# B&R Automation Studio project mappCfg
Automation Studio 4.9.3.144 SP; technology packages: mapp 5.15.0

## Configuration Config1

CPU X20CP3585, AutomationRuntime D4.90, Build 4.1.2, Safety 0.0, Vc V4.72.6

### Task classes (Cpu.sw)
```
Cyclic#4:
  MpLinkTest <- (binary)
Cyclic#8:
  MpCfgTest <- MpCfgTest.prg
Binaries: FWRules, udbdef, arsvcreg, TCData, User, arconfig, Role, Config, iomap, asfw, ashwac, ashwd, sysconf
Libraries: MpCom, MpBase, MpCfg, FileIO, runtime, astime, asieccon, AsBrStr, IecCheck, sys_lib, MpUserX
```

### Hardware
```
X20CP3585 : X20CP3585 v1.10.0.0
  Connector IF2:
    ActivateDevice = 1
  ConfigurationID = mappLink_Config1
  FtpUser1
  FtpUsername1 = bur
  FtpUserPassword1 = 9h9s1YQ4rmHMniR3mwrIYznV2yRb7wj1AtHiJ/RHOmI=  // bur
  FtpUserSalt1 = llDQoh2a
  FTPAccessRight1 = 0
  FTPMSPartition1 = SYSTEM
```

### Config.mpdatabasecore - X20CP3585/mappServices/Config.mpdatabasecore
```
Element gDatabaseCore (Type=mpdatabasecore)
  mapp.Database.Core:
    Name = brdatabase
    UserName = br
    Password = bandr
    IPAddress  // IPv4 address of the database script
    PortNumber = 85  // SQL port number of the database script
    DBQueries:
      [0]:
        Name = RecipeLoad
        Type:
          Select:
            Columns:
              PV = ::Recipe.DATA
          From = dbo.brtable
          Where:
            [0]:
              Column = product_name
              Operator = eq
              CompareTo:
                Value = {&pv[Recipe.PAR.RecipeName]}
      [1]:
        Name = RecipeSave
        Type:
          1TypeName = UPDATE
          Where:
            [0]:
              Column = product_name
              Operator = eq
              CompareTo:
                Value = {&pv[Recipe.PAR.RecipeName]}
      [2]:
        Name = RecipeDelete
        Type:
          1TypeName = DELETE
          Where:
            [0]:
              Column = product_name
              Operator = eq
              CompareTo:
                Value = {&pv[Recipe.PAR.RecipeName]}
      [3]:
        Name = RecipeNew
        Type:
          1TypeName = INSERT
      [4]:
        Name = RecipeList
        Type:
          1TypeName = Custom
```

### Config_1.mpuserx - X20CP3585/mappServices/Config_1.mpuserx
```
Element UserMgmtX (Type=mpuserx)
  ServerSettings:
    Server:
      AdditionalUserData:
        [0] = mail
        [1] = telephoneNumber
  Users:
    DefUser#1:
      id = Anonymous
      name = Nobody
    DefUser#2:
      id = John
      name = John Doe
    DefUser#3:
      id = Jane
      name = Jane Doe
```

## Logical view

Binary libraries used (declarations not repeated): operator, runtime, astime, AsIecCon, FileIO, AsBrStr, IecCheck, sys_lib, MpCom, MpBase, MpUserX 5.15.0

### Package Logical/Libraries - Global libraries

### Library Logical/Libraries/MpCfg (IEC)

#### Types.typ - Exported data types
```iecst
TYPE
	MpCfgInfoType : 	STRUCT
		state : MpCfgStateType;
		DevLink_1 : DevLink;
		FileOpen_1 : FileOpen;
		FileRead_1 : FileRead;
		FileWrite_1 : FileWrite;
		FileClose_1 : FileClose;
		MpComConfigManager_1 : MpComConfigManager;
		Buffer : ARRAY[0..MpCfgMaxBufferSize]OF USINT;
		NodeName : STRING[MpCfgMaxNameSize];
		NodeValue : STRING[MpCfgMaxValueSize];
		offset1 : DINT;
		offset2 : DINT;
		len : DINT;
		tmpStr1 : STRING[MpCfgMaxNameSize];
		tmpStr2 : STRING[MpCfgMaxNameSize];
	END_STRUCT;
	MpCfgStateType :
		(
		stateWait,
		stateDevLink,
		stateExport,
		stateOpen,
		stateRead,
		stateWrite,
		stateClose,
		stateFindData,
		stateInsertData,
		stateError
		);
END_TYPE
```

#### Constants.var - Exported constants
```iecst
(*Buffer and variable sizes*)
VAR CONSTANT
	MpCfgMaxBufferSize : UINT := 10000;
	MpCfgMaxNameSize : UINT := 200;
	MpCfgMaxValueSize : UINT := 200;
END_VAR
(*Error numbers*)
VAR CONSTANT
	MpCfgBufferSizeExceeded : DINT := 10001;
	MpCfgDataTypeSizeExceeded : DINT := 10002;
	MpCfgValueSizeExceeded : DINT := 10003;
	MpCfgGroupNotFound0 : DINT := 10010;
	MpCfgGroupNotFound1 : DINT := 10011;
	MpCfgGroupNotFound2 : DINT := 10012;
	MpCfgGroupNotFound3 : DINT := 10013;
	MpCfgGroupNotFound4 : DINT := 10014;
	MpCfgGroupNotFound5 : DINT := 10015;
	MpCfgGroupNotFound6 : DINT := 10016;
	MpCfgGroupNotFound7 : DINT := 10017;
	MpCfgGroupNotFound8 : DINT := 10018;
	MpCfgGroupNotFound9 : DINT := 10019;
	MpCfgParaNotFound : DINT := 10020;
	MpCfgTypeNotFound : DINT := 10021;
	MpCfgValueNotFound : DINT := 10022;
	MpCfgParaNameEmpty : DINT := 10030;
	MpCfgMpLinkEmpty : DINT := 10031;
END_VAR
(*Read/Write constants*)
VAR CONSTANT
	MpCfgRead : BOOL := FALSE;
	MpCfgWrite : BOOL := TRUE;
END_VAR
```

#### MpCfg.fun - Exported functions and function blocks
```iecst
FUNCTION_BLOCK MpCfgRW
	VAR_INPUT
		MpLink : {REDUND_UNREPLICABLE} MpComIdentType;
		Enable : BOOL;
		ReadWrite : BOOL;
		ErrorReset : BOOL;
		ParaName : STRING[MpCfgMaxNameSize];
		ParaValue : STRING[MpCfgMaxValueSize];
	END_VAR
	VAR_OUTPUT
		Active : BOOL;
		Error : BOOL;
		StatusID : DINT;
		CommandDone : BOOL;
		DataType : STRING[50];
		Value : STRING[MpCfgMaxValueSize];
	END_VAR
	VAR
		Info : MpCfgInfoType;
	END_VAR
END_FUNCTION_BLOCK

FUNCTION FindInMem : DINT
	VAR_INPUT
		data1 : UDINT;
		len1 : UDINT;
		data2 : UDINT;
		len2 : UDINT;
		direction : BOOL;
	END_VAR
	VAR
		idx : UDINT;
	END_VAR
END_FUNCTION

FUNCTION ReplaceString : BOOL
	VAR_INPUT
		dataSTR : UDINT;
		searchSTR : UDINT;
		replaceSTR : UDINT;
		first : BOOL;
	END_VAR
	VAR
		idx : UDINT;
	END_VAR
END_FUNCTION
```

#### MpCfg.st
```iecst
// -------------------------------------------------------------------------
// Read mapp configuration parameter
// -------------------------------------------------------------------------
FUNCTION_BLOCK MpCfgRW
	// Abort command
	IF EDGENEG(Enable) THEN
		// Close file if it was already opened
		IF Info.state >= stateOpen AND Info.state <> stateError THEN
			Info.state := stateClose;
		END_IF
	END_IF

	// -------------------------------------------------------------------------
	// MpLink state machine
	CASE Info.state OF
		// -------------------------------------------------------------------------
		// Wait for new command
		stateWait:
			// Reset all funtion blocks
			Info.DevLink_1.enable 				:= FALSE;
			Info.DevLink_1();
			Info.MpComConfigManager_1.Enable 	:= FALSE;
			Info.MpComConfigManager_1();
			Info.FileOpen_1.enable				:= FALSE;
			Info.FileOpen_1();
			Info.FileRead_1.enable				:= FALSE;
			Info.FileRead_1();
			Info.FileClose_1.enable				:= FALSE;
			Info.FileClose_1();

			// New command
			IF EDGEPOS(Enable) THEN
				// Make sure MpLink is not empty
				IF MpLink.Internal[0] = 0 THEN
					StatusID := MpCfgMpLinkEmpty;
					Info.state := stateError;
				ELSE
					// Make sure parameter is not empty
					IF ParaName = '' THEN
						StatusID := MpCfgParaNameEmpty;
						Info.state := stateError;
					ELSE
						// Set start values
						Active := TRUE;
						DataType := '';
						Value := '';
						brsmemset(ADR(Info.Buffer), 0, SIZEOF(Info.Buffer));
						Info.state := stateDevLink;
					END_IF
				END_IF
			ELSE
				IF NOT Enable THEN
					CommandDone := FALSE;
				END_IF
				Active := FALSE;
			END_IF
			// -------------------------------------------------------------------------
		// Link file device used for exporting data
		stateDevLink:
			Info.DevLink_1.enable 	:= TRUE;
			Info.DevLink_1.pDevice	:= ADR('MpCfgDev');
			Info.DevLink_1.pParam	:= ADR('/DEVICE=C:/');
			Info.DevLink_1();

			// Success
			IF Info.DevLink_1.status = ERR_OK OR Info.DevLink_1.status = fiERR_DEVICE_ALREADY_EXIST THEN
				Info.state := stateExport;
			// Errror
			ELSIF Info.DevLink_1.status <> ERR_FUB_BUSY THEN
				StatusID := Info.DevLink_1.status;
				Info.state := stateError;
			END_IF
		// -------------------------------------------------------------------------
		// Export mapp data
		stateExport:
			Info.MpComConfigManager_1.Enable 		:= TRUE;
			Info.MpComConfigManager_1.MpLink		:= ADR(MpLink);
			Info.MpComConfigManager_1.DeviceName 	:= ADR('MpCfgDev');
			Info.MpComConfigManager_1.FileName 		:= ADR('MpCfg.xml');
			Info.MpComConfigManager_1.Scope			:= mpCOM_CONFIG_SCOPE_COMPONENT;
			Info.MpComConfigManager_1.Export		:= TRUE;
			Info.MpComConfigManager_1.Import		:= FALSE;
			Info.MpComConfigManager_1();

			// Success
			IF Info.MpComConfigManager_1.CommandDone AND NOT Info.MpComConfigManager_1.Error THEN
				Info.state := stateOpen;
			// Errror
			ELSIF Info.MpComConfigManager_1.Error THEN
				StatusID := Info.MpComConfigManager_1.StatusID;
				Info.state := stateError;
			END_IF
		// -------------------------------------------------------------------------
		// Open mapp data
		stateOpen:
			Info.FileOpen_1.enable		:= TRUE;
			Info.FileOpen_1.pDevice 	:= ADR('MpCfgDev');
			Info.FileOpen_1.pFile		:= ADR('MpCfg.xml');
			Info.FileOpen_1.mode 		:= fiREAD_WRITE;
			Info.FileOpen_1();

			// Success
			IF Info.FileOpen_1.status = ERR_OK THEN
				IF Info.FileOpen_1.filelen > SIZEOF(Info.Buffer) THEN
					StatusID := MpCfgBufferSizeExceeded;
					Info.state := stateError;
				ELSE
					Info.state := stateRead;
				END_IF
			// Errror
			ELSIF Info.FileOpen_1.status <> ERR_FUB_BUSY THEN
				StatusID := Info.FileOpen_1.status;
				Info.state := stateError;
			END_IF

		// -------------------------------------------------------------------------
		// Read mapp data file
		stateRead:
			Info.FileRead_1.enable		:= TRUE;
			Info.FileRead_1.ident		:= Info.FileOpen_1.ident;
			Info.FileRead_1.len			:= Info.FileOpen_1.filelen;
			Info.FileRead_1.pDest		:= ADR(Info.Buffer);
			Info.FileRead_1();

			// Success
			IF Info.FileRead_1.status = ERR_OK THEN
				// Find group id first
				IF ADR(GroupArray) <> 0 THEN
					// Make sure array has at least one entry
					IF GroupArray.Item[0] <> '' THEN
						Info.idx := 0;
						Info.DataOffset1 := 0;
						Info.state := stateFindGroup;
					// Find unique parameter
					ELSE
						Info.state := stateFindData;
					END_IF
				// Find unique parameter
				ELSE
					Info.state := stateFindData;
				END_IF
			// Errror
			ELSIF Info.FileRead_1.status <> ERR_FUB_BUSY THEN
				StatusID := Info.FileRead_1.status;
				Info.state := stateError;
			END_IF

		// -------------------------------------------------------------------------
		// Write mapp data file
		stateWrite:
			Info.FileWrite_1.enable		:= TRUE;
			Info.FileWrite_1.ident		:= Info.FileOpen_1.ident;
			Info.FileWrite_1.len		:= Info.FileLen;
			Info.FileWrite_1.pSrc		:= ADR(Info.Buffer);
			Info.FileWrite_1();

			// Success
			IF Info.FileWrite_1.status = ERR_OK THEN
				Info.state := stateClose;
			// Errror
			ELSIF Info.FileWrite_1.status <> ERR_FUB_BUSY THEN
				StatusID := Info.FileWrite_1.status;
				Info.state := stateError;
			END_IF

		// -------------------------------------------------------------------------
		// Find group data
		stateFindGroup:
			// Prepare group string
			Info.tmpStr1 := '<Group ID="';
			brsstrcat(ADR(Info.tmpStr1), ADR(GroupArray.Item[Info.idx]));
			brsstrcat(ADR(Info.tmpStr1), ADR('"'));
			// Find property string
			Info.DataOffset1 := Info.DataOffset1+FindInMem(ADR(Info.Buffer)+Info.DataOffset1, Info.FileOpen_1.filelen, ADR(Info.tmpStr1), brsstrlen(ADR(Info.tmpStr1)), FALSE);

			// Found group string
			IF Info.DataOffset1 > -1 THEN
				// Find next group name
				IF Info.idx < SIZEOF(GroupArray)/SIZEOF(GroupArray.Item[0]) THEN
					Info.idx := Info.idx + 1;
					IF GroupArray.Item[Info.idx] = '' THEN
						Info.state := stateFindData;
					END_IF
				// Group was not found
				ELSE
					StatusID := MpCfgGroupNotFound0+Info.idx;
					Info.state := stateError;
				END_IF
			// Group was not found
			ELSE
				StatusID := MpCfgGroupNotFound0+Info.idx;
				Info.state := stateError;
			END_IF
		// -------------------------------------------------------------------------
		// Find data
		stateFindData:
			// Prepare property string
			Info.tmpStr1 := '<Property ID="';
			brsstrcat(ADR(Info.tmpStr1), ADR(ParaName));
			brsstrcat(ADR(Info.tmpStr1), ADR('"'));
			// Find property string
			Info.DataOffset1 := Info.DataOffset1+FindInMem(ADR(Info.Buffer)+Info.DataOffset1, Info.FileOpen_1.filelen, ADR(Info.tmpStr1), brsstrlen(ADR(Info.tmpStr1)), FALSE);

			// Found parameter string
			IF Info.DataOffset1 > -1 THEN
				// Prepare data type start string
				Info.tmpStr1 := 'DataType="';
				// Find data type string start
				Info.DataOffset2 := brsstrlen(ADR(Info.tmpStr1))+FindInMem(ADR(Info.Buffer)+Info.DataOffset1, Info.FileOpen_1.filelen, ADR(Info.tmpStr1), brsstrlen(ADR(Info.tmpStr1)), FALSE);

				// Found data type start
				IF Info.DataOffset2 > -1 THEN
					// Prepare data type end string
					Info.tmpStr1 := '"';
					// Find data type string
					Info.DataLen := FindInMem(ADR(Info.Buffer)+Info.DataOffset1+Info.DataOffset2, Info.FileOpen_1.filelen, ADR(Info.tmpStr1), brsstrlen(ADR(Info.tmpStr1)), FALSE);

					// Found data type end, copy data to output
					IF Info.DataLen > -1 THEN
						brsmemset(ADR(DataType), 0, SIZEOF(DataType));
						brsmemcpy(ADR(DataType), ADR(Info.Buffer)+Info.DataOffset1+Info.DataOffset2, Info.DataLen);

						// Prepare value start string
						Info.tmpStr1 := 'Value="';
						// Find data type string start
						Info.DataOffset2 := brsstrlen(ADR(Info.tmpStr1))+FindInMem(ADR(Info.Buffer)+Info.DataOffset1, Info.FileOpen_1.filelen, ADR(Info.tmpStr1), brsstrlen(ADR(Info.tmpStr1)), FALSE);

						// Found value start
						IF Info.DataOffset2 > -1 THEN
							// Prepare value end string
							Info.tmpStr1 := '"';
							// Find value end string
							Info.DataLen := FindInMem(ADR(Info.Buffer)+Info.DataOffset1+Info.DataOffset2, Info.FileOpen_1.filelen, ADR(Info.tmpStr1), brsstrlen(ADR(Info.tmpStr1)), FALSE);

							// Found value end, copy data to output
							IF Info.DataLen > -1 THEN
								brsmemset(ADR(Value), 0, SIZEOF(Value));
								brsmemcpy(ADR(Value), ADR(Info.Buffer)+Info.DataOffset1+Info.DataOffset2, Info.DataLen);

								// Finish when command is reading
								IF ReadWrite = MpCfgRead THEN
									Info.state := stateClose;
								// Insert new data in next step
								ELSE
									Info.state := stateInsertData;
								END_IF
							// Value end was not found
							ELSE
								StatusID := MpCfgValueNotFound;
								Info.state := stateError;
							END_IF
						// Value start was not found
						ELSE
							StatusID := MpCfgValueNotFound;
							Info.state := stateError;
						END_IF
					// Data type end was not found
					ELSE
						StatusID := MpCfgTypeNotFound;
						Info.state := stateError;
					END_IF
				// Data type end was not found
				ELSE
					StatusID := MpCfgTypeNotFound;
					Info.state := stateError;
				END_IF
			// Parameter name was not found
			ELSE
				StatusID := MpCfgParaNotFound;
				Info.state := stateError;
			END_IF

		// -------------------------------------------------------------------------
		// Insert new data
		stateInsertData:
			// Calculate start address for value
			Info.DataOffset3 := ADR(Info.Buffer)+Info.DataOffset1+Info.DataOffset2;
			// Calculate remaining data
			Info.DataLen := Info.FileOpen_1.filelen-(Info.DataOffset1+Info.DataOffset2);

			brsmemmove(Info.DataOffset3+brsstrlen(ADR(ParaValue)), Info.DataOffset3+brsstrlen(ADR(Value)), Info.DataLen-brsstrlen(ADR(Value))+1);
			brsmemcpy(Info.DataOffset3, ADR(ParaValue), brsstrlen(ADR(ParaValue)));

			// New value is shorter than old
			IF brsstrlen(ADR(Value)) >= brsstrlen(ADR(ParaValue)) THEN
				Info.FileLen := Info.FileOpen_1.filelen;
				// Fill taling memory with LF if new data is smaller than old
				brsmemset(ADR(Info.Buffer)+Info.FileLen, 10, brsstrlen(ADR(Value))-brsstrlen(ADR(ParaValue)));
			// New value is larger than old
			ELSE
				Info.FileLen := Info.FileOpen_1.filelen+(brsstrlen(ADR(ParaValue))-brsstrlen(ADR(Value)));
			END_IF

			Info.state := stateWrite;

		// -------------------------------------------------------------------------
		// Close mapp data file
		stateClose:
			Info.FileClose_1.enable		:= TRUE;
			Info.FileClose_1.ident		:= Info.FileOpen_1.ident;
			Info.FileClose_1();

			// Success
			IF Info.FileClose_1.status = ERR_OK THEN
				Info.FileOpen_1.enable := FALSE;

				// When we read it ends here
				IF ReadWrite = MpCfgRead THEN
					Active := FALSE;
					CommandDone := TRUE;
					Info.state := stateWait;
				// Import new configuration
				ELSE
					Info.state := stateImport;
				END_IF
				// Errror
			ELSIF Info.FileClose_1.status <> ERR_FUB_BUSY THEN
				StatusID := Info.FileClose_1.status;
				Info.state := stateError;
			END_IF

		// -------------------------------------------------------------------------
		// Import mapp data
		stateImport:
			Info.MpComConfigManager_1.Enable 		:= TRUE;
			Info.MpComConfigManager_1.MpLink		:= ADR(MpLink);
			Info.MpComConfigManager_1.DeviceName 	:= ADR('MpCfgDev');
			Info.MpComConfigManager_1.FileName 		:= ADR('MpCfg.xml');
			Info.MpComConfigManager_1.Scope			:= mpCOM_CONFIG_SCOPE_COMPONENT;
			Info.MpComConfigManager_1.Export		:= FALSE;
			Info.MpComConfigManager_1.Import		:= TRUE;
			Info.MpComConfigManager_1();

			// Success
			IF Info.MpComConfigManager_1.CommandDone AND NOT Info.MpComConfigManager_1.Error THEN
				Active := FALSE;
				CommandDone := TRUE;
				Info.state := stateWait;
			// Errror
			ELSIF Info.MpComConfigManager_1.Error THEN
				StatusID := Info.MpComConfigManager_1.StatusID;
				Info.state := stateError;
			END_IF

		// -------------------------------------------------------------------------
		// Error state
		stateError:
			// Close file when it is open
			IF Info.FileOpen_1.enable THEN
				Info.FileClose_1.enable	:= TRUE;
				Info.FileClose_1.ident	:= Info.FileOpen_1.ident;
				Info.FileClose_1();
			END_IF

			// Set flags
			Active := FALSE;
			Error := TRUE;
			CommandDone := TRUE;

			// Wait for error reset
			IF ErrorReset THEN
				StatusID := 0;
				Error := FALSE;
				Info.state := stateWait;
			END_IF
	END_CASE;

	ErrorReset := FALSE;
END_FUNCTION_BLOCK
```

#### LocalFunctions.st
```iecst
//******************************************************************************************************
// Find second data in first data
//******************************************************************************************************
FUNCTION FindInMem
	FindInMem := -1;
	IF (len1 > len2) THEN
		IF(direction) THEN
			idx := len1 - len2;
			WHILE(idx > 0) DO
				IF (brsmemcmp(data1 + idx, data2, len2) = 0) THEN
					FindInMem := idx;
					EXIT;
				END_IF
				idx := idx - 1;
			END_WHILE;
		ELSE
			FOR idx:=0 TO len1 - len2 DO
				IF (brsmemcmp(data1 + idx, data2, len2) = 0) THEN
					FindInMem := idx;
					EXIT;
				END_IF
			END_FOR;
		END_IF
	END_IF
END_FUNCTION

//******************************************************************************************************
// Find and replace string
//******************************************************************************************************
FUNCTION ReplaceString
	IF (brsstrlen(dataSTR) >= brsstrlen(searchSTR)) THEN
		FOR idx:=0 TO brsstrlen(dataSTR) - brsstrlen(searchSTR) DO
			IF (brsmemcmp(dataSTR + idx, searchSTR, brsstrlen(searchSTR)) = 0) THEN
				// Move data around
				brsmemmove(dataSTR + idx + brsstrlen(replaceSTR), dataSTR + idx + brsstrlen(searchSTR), brsstrlen(dataSTR) - brsstrlen(searchSTR) + 1);
				brsmemcpy(dataSTR + idx, replaceSTR, brsstrlen(replaceSTR));
				// Set found flag and exit if only one hit is needed
				ReplaceString := TRUE;
				IF(first) THEN
					EXIT;
				END_IF
				// Correct index for next search
				IF(brsstrlen(replaceSTR) > 0) THEN
					idx := idx + brsstrlen(replaceSTR);
				END_IF
				idx := idx - 1;
				// Exit if no data is left
				IF (brsstrlen(dataSTR) = 0 OR brsstrlen(dataSTR) < brsstrlen(searchSTR)) THEN
					EXIT;
				END_IF
			END_IF
		END_FOR;
	END_IF
END_FUNCTION
```

### Library Logical/Libraries/MpLink (IEC)

#### Types.typ - Exported data types
```iecst
TYPE
	MpLinkInfoType : 	STRUCT
		state : MpLinkStateType;
		DevLink_01 : DevLink;
		MpComConfigManager_01 : MpComConfigManager;
	END_STRUCT;
	MpLinkStateType :
		(
		stateWait,
		stateDevLink,
		stateExport
		);
END_TYPE
```

#### MpLink.fun - Exported functions and function blocks
```iecst
FUNCTION_BLOCK MpReadLink
	VAR_INPUT
		MpLink : REFERENCE TO MpComIdentType;
		Enable : BOOL;
		ErrorReset : BOOL;
		ParaName : STRING[80];
	END_VAR
	VAR_OUTPUT
		Active : BOOL;
		Error : BOOL;
		StatusID : DINT;
		CommandDone : BOOL;
	END_VAR
	VAR
		Info : MpLinkInfoType;
	END_VAR
END_FUNCTION_BLOCK
```

#### MpReadLink.st
```iecst
// -------------------------------------------------------------------------
// Read mapp configuration parameter
// -------------------------------------------------------------------------
FUNCTION_BLOCK MpReadLink
	// -------------------------------------------------------------------------
	// MpLink state machine
	CASE Info.state OF
		// -------------------------------------------------------------------------
		// Wait for new command
		stateWait:
			IF Enable THEN
				Active := TRUE;
				Info.state := stateDevLink;
			ELSE
				Active := FALSE;
			END_IF
		// -------------------------------------------------------------------------
		// Link file device used for exporting data
		stateDevLink:
			Info.DevLink_01.enable 	:= TRUE;
			Info.DevLink_01.pDevice := ADR('MpLinkDev');
			Info.DevLink_01.pParam	:= ADR('/DEVICE=C:/');
			Info.DevLink_01();

			// Success
			IF Info.DevLink_01.status = ERR_OK THEN
				Info.state := stateExport;
			// Errror
			ELSIF Info.DevLink_01.status <> ERR_FUB_BUSY THEN
			END_IF
		// -------------------------------------------------------------------------
		// Export mapp data
		stateExport:
			Info.MpComConfigManager_01.Enable 		:= TRUE;
			Info.MpComConfigManager_01.DeviceName 	:= ADR('MpLinkDev');
			Info.MpComConfigManager_01.FileName 	:= ADR('MpLink.xml');
			Info.MpComConfigManager_01.Scope		:= mpCOM_CONFIG_SCOPE_COMPONENT;
			Info.MpComConfigManager_01.Export		:= TRUE;
			Info.MpComConfigManager_01();

			IF Info.MpComConfigManager_01.CommandDone THEN
			END_IF
	END_CASE;
END_FUNCTION_BLOCK
```

### Program Logical/MpCfgTest (IEC)

#### Variables.var
```iecst
VAR
	mappReadUnique : BOOL; (*Read unique value*)
	mappReadGroup : BOOL; (*Read not unique value*)
	mappWriteUnique : BOOL; (*Write unique value*)
	mappWriteGroup : BOOL; (*Write not unique value*)
	GroupArray : MpCfgGroupArray; (*Group array used for not unique values*)
	MpCfgRW_01 : MpCfgRW; (*Functionblock for mapp configuration read/write*)
END_VAR
```

#### Main.st
```iecst
PROGRAM _CYCLIC

	// Read unique mapp configuration parameter
	IF mappReadUnique THEN
		MpCfgRW_01.Enable 		:= TRUE;
		MpCfgRW_01.MpLink 		:= gDatabaseCore;
		MpCfgRW_01.ReadWrite 	:= MpCfgRead;
		MpCfgRW_01.ParaName 	:= 'IPAddress';
		MpCfgRW_01.GroupArray	:= 0;

		IF MpCfgRW_01.CommandDone THEN
			MpCfgRW_01.Enable := FALSE;
			mappReadUnique := FALSE;
		END_IF
	END_IF

	// Read mapp configuration parameter with additional group information
	IF mappReadGroup THEN
		// Group array definition
		GroupArray.Item[0] := 'mapp.Database.Core';
		GroupArray.Item[1] := 'DBQueries';
		GroupArray.Item[2] := '[1]';
		GroupArray.Item[3] := 'Where';
		GroupArray.Item[4] := '[0]';

		MpCfgRW_01.Enable 		:= TRUE;
		MpCfgRW_01.MpLink 		:= gDatabaseCore;
		MpCfgRW_01.ReadWrite 	:= MpCfgRead;
		MpCfgRW_01.ParaName 	:= 'Column';
		MpCfgRW_01.GroupArray	:= ADR(GroupArray);

		IF MpCfgRW_01.CommandDone THEN
			MpCfgRW_01.Enable := FALSE;
			mappReadGroup := FALSE;
		END_IF
	END_IF

	// Write unique mapp configuration parameter
	IF mappWriteUnique THEN
		MpCfgRW_01.Enable 		:= TRUE;
		MpCfgRW_01.MpLink 		:= gDatabaseCore;
		MpCfgRW_01.ReadWrite 	:= MpCfgWrite;
		MpCfgRW_01.ParaName 	:= 'IPAddress';
		MpCfgRW_01.ParaValue 	:= '192.168.0.1';
		MpCfgRW_01.GroupArray	:= 0;

		IF MpCfgRW_01.CommandDone THEN
			MpCfgRW_01.Enable := FALSE;
			mappWriteUnique := FALSE;
		END_IF
	END_IF

	// Write mapp configuration parameter with additional group information
	IF mappWriteGroup THEN
		// Group array definition
		GroupArray.Item[0] := 'mapp.Database.Core';
		GroupArray.Item[1] := 'DBQueries';
		GroupArray.Item[2] := '[1]';
		GroupArray.Item[3] := 'Where';
		GroupArray.Item[4] := '[0]';

		MpCfgRW_01.Enable 		:= TRUE;
		MpCfgRW_01.MpLink 		:= gDatabaseCore;
		MpCfgRW_01.ReadWrite 	:= MpCfgWrite;
		MpCfgRW_01.ParaName 	:= 'Column';
		MpCfgRW_01.ParaValue 	:= 'product_group';
		MpCfgRW_01.GroupArray	:= ADR(GroupArray);

		IF MpCfgRW_01.CommandDone THEN
			MpCfgRW_01.Enable := FALSE;
			mappWriteGroup := FALSE;
		END_IF
	END_IF

	MpCfgRW_01();

END_PROGRAM
```

### Program Logical/MpLinkTest

#### Variables.var
```iecst
VAR
	Read : BOOL;
	MpReadLink_01 : MpReadLink;
END_VAR
```

#### Main.st
```iecst
PROGRAM _INIT

END_PROGRAM

PROGRAM _CYCLIC
	IF Read THEN
		MpReadLink_01.Enable := TRUE;
		MpReadLink_01.MpLink := ADR(gDatabaseCore);
	END_IF

END_PROGRAM
```

Listed in the project but not available here: Logical/Global.typ, Logical/Global.var, Logical/Libraries/MpLink/Constants.var
